Fanuc KAREL source: ko00067.KL

PROGRAM KO00067
%STACKSIZE=65535
%PRIORITY=65535
%NOLOCKGROUP
VAR
P1 : XYZWPREXT
P2 : POSITION
F : BOOLEAN
OUT : XYZWPREXT
BEGIN
F=TRUE
OUT=MIRROR(P1,P2,F)
END KO00067
